KUKA KRL program: edge_1_right_stm.src, edge_1_right_stm.dat

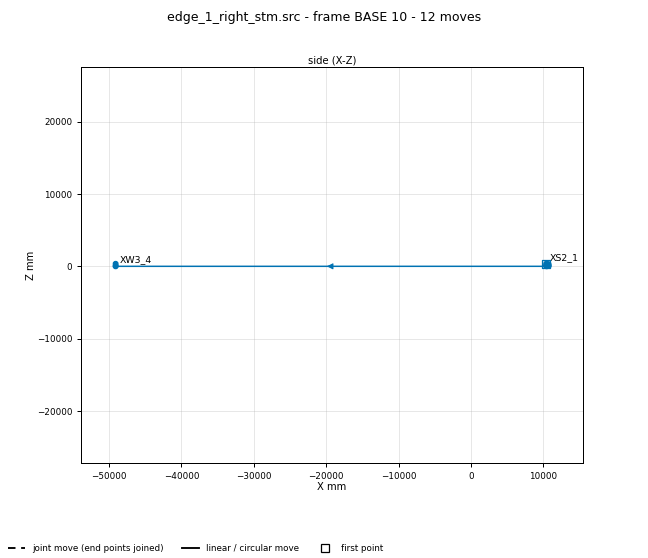
[picture p0: tool path of edge_1_right_stm.src in frame BASE 10, 12 of 12 moves have a stored position in this frame; points joined in program order, loops and branches not executed]
--- edge_1_right_stm.src ---
&ACCESS RVP
&REL 45
&PARAM EDITMASK = *
&PARAM DISKPATH = KRC:\R1\Program
DEF edge_1_right_stm( )
;FOLD INI;%{PE}
  ;FOLD BASISTECH INI
    GLOBAL INTERRUPT DECL 3 WHEN $STOPMESS==TRUE DO IR_STOPM ( )
    INTERRUPT ON 3
    BAS (#INITMOV,0 )
  ;ENDFOLD (BASISTECH INI)
  ;FOLD USER INI
    ;Make your modifications here

  ;ENDFOLD (USER INI)
;ENDFOLD (INI)
TS_CorrOff()
;FOLD PTP S2_1 Vel= 100 % PDATW1_1 Tool[1] Base[10] ;%{PE}%R 8.3.34,%MKUKATPBASIS,%CMOVE,%VPTP,%P 1:PTP, 2:S2_1, 3:C_DIS, 5:100, 7:PDATS2_1
$BWDSTART = FALSE
PDAT_ACT=PPDATS2_1
FDAT_ACT=FS2_1
BAS(#PTP_PARAMS,100)
SET_CD_PARAMS (0)
PTP XS2_1 C_DIS
;ENDFOLD

;FOLD LIN S2_2 Vel= 0.06 m/s CPDATS2_2 TouchSense SEARCH VIA S2_3 CDS2_2 SPS2_2 Tool[1] Base[10] ;%{PE}
;FOLD Parameters ;%{h}
;Params IlfProvider=kukaroboter.touchsense.searchlin; Kuka.PointName=S2_2; Kuka.BlendingEnabled=False; Kuka.MoveDataName=CPDATS2_2; Kuka.VelocityPath=0.06; Kuka.MovementParameterFieldEnabled=True; MoveType=LIN
;FOLD Parameters TouchSense ;%{h}
;Params TouchSense.SearchViaPoint=S2_3;TouchSense.ReferenceMove=CDS2_2;TouchSense.SeachParam=SPS2_2
;ENDFOLD
;ENDFOLD
$BWDSTART = FALSE
LDAT_ACT=LCPDATS2_2
FDAT_ACT=FS2_2
BAS(#CP_PARAMS,0.06)
SET_CD_PARAMS (0)
LIN XS2_2 C_DIS C_DIS
TS_InitMovement($POS_ACT, XS2_3, ZSPS2_2)
TS_ManMoveToVia(XS2_3)
TS_Search(XS2_3, ZSPS2_2, VCDS2_2)
TS_SetCorrData(ZSPS2_2, VCDS2_2)
;ENDFOLD

;FOLD TouchSense Corr 1 CDS2_2;%{E}
;FOLD Parameters Corr 1D ;%{h}
;Params IlfProvider=KukaRoboter.TouchSense.Correction1D;Correction1D=CDS2_2
;ENDFOLD
TS_BC6DCalc(VCDS2_2, TSg_CD0, TSg_CD0, TSg_CD0, TSg_CD0, TSg_CD0)
;ENDFOLD

;FOLD LIN S2_4 Vel= 0.06 m/s CPDATS2_4 TouchSense SEARCH VIA S2_5 CDS2_4 SPS2_4 Tool[1] Base[10] ;%{PE}
;FOLD Parameters ;%{h}
;Params IlfProvider=kukaroboter.touchsense.searchlin; Kuka.PointName=S2_4; Kuka.BlendingEnabled=False; Kuka.MoveDataName=CPDATS2_4; Kuka.VelocityPath=0.06; Kuka.MovementParameterFieldEnabled=True; MoveType=LIN
;FOLD Parameters TouchSense ;%{h}
;Params TouchSense.SearchViaPoint=S2_5;TouchSense.ReferenceMove=CDS2_4;TouchSense.SeachParam=SPS2_4
;ENDFOLD
;ENDFOLD
$BWDSTART = FALSE
LDAT_ACT=LCPDATS2_4
FDAT_ACT=FS2_4
BAS(#CP_PARAMS,0.06)
SET_CD_PARAMS (0)
LIN XS2_4 C_DIS C_DIS
TS_InitMovement($POS_ACT, XS2_5, ZSPS2_4)
TS_ManMoveToVia(XS2_5)
TS_Search(XS2_5, ZSPS2_4, VCDS2_4)
TS_SetCorrData(ZSPS2_4, VCDS2_4)
;ENDFOLD

;FOLD TouchSense Corr 2 CDS2_2 CDS2_4;%{E}
;FOLD Parameters Corr 2D ;%{h}
;Params IlfProvider=KukaRoboter.TouchSense.Correction2D;Correction1D=CDS2_2;Correction2D=CDS2_4
;ENDFOLD
TS_BC6DCalc(VCDS2_2, TSg_CD0, TSg_CD0, VCDS2_4, TSg_CD0, TSg_CD0)
;ENDFOLD

;FOLD LIN S2_6 Vel= 0.06 m/s CPDATS1_2 Tool[1] Base[10] ;%{PE}%R 8.3.34,%MKUKATPBASIS,%CMOVE,%VLIN,%P 1:LIN, 2:S2_6, 3:, 5:0.06, 7:CPDATS2_6
$BWDSTART = FALSE
LDAT_ACT=LCPDATS2_6
FDAT_ACT=FS2_6
BAS(#CP_PARAMS,0.06)
SET_CD_PARAMS (0)
LIN XS2_6 C_DIS C_DIS
;ENDFOLD

;FOLD LIN S2_7 Vel= 0.02 m/s CPDATS2_7 TouchSense SEARCH VIA S2_8 CDS2_7 SPS2_7 Tool[1] Base[10] ;%{PE}
;FOLD Parameters ;%{h}
;Params IlfProvider=kukaroboter.touchsense.searchlin; Kuka.PointName=S2_7; Kuka.BlendingEnabled=False; Kuka.MoveDataName=CPDATS2_7; Kuka.VelocityPath=0.02; Kuka.MovementParameterFieldEnabled=True; MoveType=LIN
;FOLD Parameters TouchSense ;%{h}
;Params TouchSense.SearchViaPoint=S2_8;TouchSense.ReferenceMove=CDS2_7;TouchSense.SeachParam=SPS2_7
;ENDFOLD
;ENDFOLD
$BWDSTART = FALSE
LDAT_ACT=LCPDATS2_7
FDAT_ACT=FS2_7
BAS(#CP_PARAMS,0.02)
SET_CD_PARAMS (0)
LIN XS2_7 C_DIS C_DIS
TS_InitMovement($POS_ACT, XS2_8, ZSPS2_7)
TS_ManMoveToVia(XS2_8)
TS_Search(XS2_8, ZSPS2_7, VCDS2_7)
TS_SetCorrData(ZSPS2_7, VCDS2_7)
;ENDFOLD

;FOLD TouchSense Corr 3 CDS2_2 CDS2_4 CDS2_7;%{E}
;FOLD Parameters Corr 3D ;%{h}
;Params IlfProvider=KukaRoboter.TouchSense.Correction3D;Correction1D=CDS2_2;Correction2D=CDS2_4;Correction3D=CDS2_7
;ENDFOLD
TS_BC6DCalc(VCDS2_2, TSg_CD0, TSg_CD0, VCDS2_4, TSg_CD0, VCDS2_7)
;ENDFOLD

;FOLD LIN S2_9 Vel= 0.1 m/s CPDATS1_2 Tool[1] Base[10] ;%{PE}%R 8.3.34,%MKUKATPBASIS,%CMOVE,%VLIN,%P 1:LIN, 2:S2_9, 3:, 5:0.1, 7:CPDATS2_9
$BWDSTART = FALSE
LDAT_ACT=LCPDATS2_9
FDAT_ACT=FS2_9
BAS(#CP_PARAMS,0.1)
SET_CD_PARAMS (0)
LIN XS2_9 C_DIS C_DIS
;ENDFOLD

;FOLD PTP W3_1 Vel= 100 % PDATW1_1 Tool[1] Base[10] ;%{PE}%R 8.3.34,%MKUKATPBASIS,%CMOVE,%VPTP,%P 1:PTP, 2:W3_1, 3:C_DIS, 5:100, 7:PDATW3_1
$BWDSTART = FALSE
PDAT_ACT=PPDATW3_1
FDAT_ACT=FW3_1
BAS(#PTP_PARAMS,100)
SET_CD_PARAMS (0)
PTP XW3_1 C_DIS
;ENDFOLD

;FOLD LIN W3_2 Vel= 0.2 m/s CPDATS1_2 Tool[1] Base[10] ;%{PE}%R 8.3.34,%MKUKATPBASIS,%CMOVE,%VLIN,%P 1:LIN, 2:W3_2, 3:, 5:0.2, 7:CPDATW3_2
$BWDSTART = FALSE
LDAT_ACT=LCPDATW3_2
FDAT_ACT=FW3_2
BAS(#CP_PARAMS,0.2)
SET_CD_PARAMS (0)
LIN XW3_2 C_DIS C_DIS
;ENDFOLD

custom_sync('hFAFA0000', 'hffff0000', 250)

;FOLD ARCON WDATW3_3 LIN W3_3 Vel= 0.1 m/s CPDATW8_4 Tool[1] Base[10];%{PE}
;FOLD Parameters ;%{h}
;Params IlfProvider=kukaroboter.arctech.arconlin; Kuka.PointName=W3_3; Kuka.BlendingEnabled=False; Kuka.MoveDataName=CPDATW3_3; Kuka.VelocityPath=0.1; Kuka.CurrentCDSetIndex=0; Kuka.MovementParameterFieldEnabled=True; ArcTech.WdatVarName=WDATW3_3
;ENDFOLD
$BWDSTART = FALSE
LDAT_ACT = LCPDATW3_3
FDAT_ACT = FW3_3
BAS(#CP_PARAMS,0.1)
SET_CD_PARAMS (0)
TRIGGER WHEN DISTANCE = 1 DELAY = ArcGetDelay(#PreDefinition, WDATW3_3) DO ArcMainNG(#PreDefinition, WDATW3_3, WW3_3) PRIO = -1
TRIGGER WHEN PATH = ArcGetPath(#OnTheFlyArcOn, WDATW3_3) DELAY = ArcGetDelay(#GasPreflow, WDATW3_3) DO ArcMainNG(#GasPreflow, WDATW3_3, WW3_3) PRIO = -1
TRIGGER WHEN PATH = ArcGetPath(#OnTheFlyArcOn, WDATW3_3) DELAY = 0 DO ArcMainNG(#ArcOnMoveStd, WDATW3_3, WW3_3) PRIO = -1
ArcMainNG(#ArcOnBeforeMoveStd, WDATW3_3, WW3_3)
LIN XW3_3
ArcMainNG(#ArcOnAfterMoveStd, WDATW3_3, WW3_3)
;ENDFOLD

;FOLD ARCOFF WDATW3_4 LIN W3_4 CPDATW3_4 Tool[1] Base[10];%{PE}
;FOLD Parameters ;%{h}
;Params IlfProvider=kukaroboter.arctech.arcofflin; Kuka.IsGlobalPoint=False; Kuka.PointName=W3_4; Kuka.BlendingEnabled=False; Kuka.MoveDataName=CPDATW3_4; Kuka.VelocityPath=0.0063; Kuka.CurrentCDSetIndex=0; Kuka.MovementParameterFieldEnabled=True; ArcTech.WdatVarName=WDATW3_4
;ENDFOLD
$BWDSTART = FALSE
LDAT_ACT = LCPDATW3_4
FDAT_ACT = FW3_4
BAS(#CP_PARAMS, gArcBasVelDefinition)
SET_CD_PARAMS (0)
TRIGGER WHEN PATH = ArcGetPath(#ArcOffBefore, WDATW3_4) DELAY = 0 DO ArcMainNG(#ArcOffBeforeOffStd, WDATW3_4) PRIO = -1
TRIGGER WHEN PATH = ArcGetPath(#OnTheFlyArcOff, WDATW3_4) DELAY = 0 DO ArcMainNG(#ArcOffMoveStd, WDATW3_4) PRIO = -1
ArcMainNG(#ArcOffBeforeMoveStd, WDATW3_4)
LIN XW3_4
ArcMainNG(#ArcOffAfterMoveStd, WDATW3_4)
;ENDFOLD

;FOLD LIN W3_5 Vel= 0.2 m/s CPDATS1_2 Tool[1] Base[10] ;%{PE}%R 8.3.34,%MKUKATPBASIS,%CMOVE,%VLIN,%P 1:LIN, 2:W3_5, 3:, 5:0.2, 7:CPDATW3_5
$BWDSTART = FALSE
LDAT_ACT=LCPDATW3_5
FDAT_ACT=FW3_5
BAS(#CP_PARAMS,0.2)
SET_CD_PARAMS (0)
LIN XW3_5 C_DIS C_DIS
;ENDFOLD

;FOLD LIN W3_6 Vel= 0.4 m/s CPDATS1_2 Tool[1] Base[10] ;%{PE}%R 8.3.34,%MKUKATPBASIS,%CMOVE,%VLIN,%P 1:LIN, 2:W3_6, 3:, 5:0.4, 7:CPDATW3_6
$BWDSTART = FALSE
LDAT_ACT=LCPDATW3_6
FDAT_ACT=FW3_6
BAS(#CP_PARAMS,0.4)
SET_CD_PARAMS (0)
LIN XW3_6 C_DIS C_DIS
;ENDFOLD

TS_CorrOff()
ochistka_mod()
END

--- edge_1_right_stm.dat ---
&ACCESS RVP
&REL 45
&PARAM EDITMASK = *
&PARAM DISKPATH = KRC:\R1\Program
DEFDAT  edge_1_right_stm
;FOLD EXTERNAL DECLARATIONS;%{PE}%MKUKATPBASIS,%CEXT,%VCOMMON,%P
;FOLD BASISTECH EXT;%{PE}%MKUKATPBASIS,%CEXT,%VEXT,%P
EXT  BAS (BAS_COMMAND  :IN,REAL  :IN )
DECL INT SUCCESS
;ENDFOLD (BASISTECH EXT)
;FOLD USER EXT;%{E}%MKUKATPUSER,%CEXT,%VEXT,%P
;Make your modifications here

;ENDFOLD (USER EXT)
;ENDFOLD (EXTERNAL DECLARATIONS)

DECL PDAT PPDATS2_1={VEL 100,ACC 100.0,APO_DIST 10.0,GEAR_JERK 50.0000,EXAX_IGN 0}
DECL FDAT FS2_1={TOOL_NO 1,BASE_NO 10,IPO_FRAME #BASE,POINT2[] " "}
DECL E6POS XS2_1={X 10410.0,Y 968.0,Z 366.0,A -120,B 50,C -180,S 20,T 53,E1 9363.166987703404,E2 0,E3 465.0,E4 0,E5 0,E6 0}

DECL E6POS XS2_2={X 10410.0,Y 968.0,Z 76.0,A -120,B 50,C -180,S 20,T 53,E1 9363.166987703404,E2 0,E3 465.0,E4 0,E5 0,E6 0}
DECL FDAT FS2_2={TOOL_NO 1,BASE_NO 10,IPO_FRAME #BASE,POINT2[] " ",TQ_STATE FALSE}
DECL LDAT LCPDATS2_2={VEL 0.06,ACC 100.0,APO_DIST 10.0,APO_FAC 50.0,ORI_TYP #VAR,CIRC_TYP #BASE,JERK_FAC 50.0}
DECL E6POS XS2_3={X 10410.0,Y 968.0,Z 16.0,A -120,B 50,C -180,S 20,T 53,E1 9363.166987703404,E2 0,E3 465.0,E4 0,E5 0,E6 0}
DECL FDAT FS2_3={TOOL_NO 1,BASE_NO 10,IPO_FRAME #BASE,POINT2[] " ",TQ_STATE FALSE}
DECL TSg_PCollCD_T VCDS2_2={CD_IPO_MODE #BASE,Mastered TRUE,SDir_W {X 0.0,Y 0.0,Z 0.0,A 0.0,B 0.0,C 0.0},Ref_W {X 10410.0,Y 968.0,Z 16.0,A -120,B 50,C -180},Meas_W {X 0.0,Y 0.0,Z 0.0,A 0.0,B 0.0,C 0.0},Diff_W {X 0.0,Y 0.0,Z 0.0,A 0.0,B 0.0,C 0.0},VecLenDiff_W 0.0,MEnum #CDEmpty,MC 1}
DECL TSg_SearchProperty_T ZSPS2_2={MoveType #MoveWithLin,TouchType #Single,DynamicStep #Slow,SensorNum 1,SearchDepth_Tol 150.0,bBackToStartPos TRUE}

DECL E6POS XS2_4={X 10410.0,Y 968.0,Z 76.0,A -120,B 50,C 169,S 20,T 53,E1 9416.675227415548,E2 0,E3 465.0,E4 0,E5 0,E6 0}
DECL FDAT FS2_4={TOOL_NO 1,BASE_NO 10,IPO_FRAME #BASE,POINT2[] " ",TQ_STATE FALSE}
DECL LDAT LCPDATS2_4={VEL 0.06,ACC 100.0,APO_DIST 10.0,APO_FAC 50.0,ORI_TYP #VAR,CIRC_TYP #BASE,JERK_FAC 50.0}
DECL E6POS XS2_5={X 10410.0,Y 908.0,Z 76.0,A -120,B 50,C 169,S 20,T 53,E1 9416.675227415548,E2 0,E3 465.0,E4 0,E5 0,E6 0}
DECL FDAT FS2_5={TOOL_NO 1,BASE_NO 10,IPO_FRAME #BASE,POINT2[] " ",TQ_STATE FALSE}
DECL TSg_PCollCD_T VCDS2_4={CD_IPO_MODE #BASE,Mastered TRUE,SDir_W {X 0.0,Y 0.0,Z 0.0,A 0.0,B 0.0,C 0.0},Ref_W {X 10410.0,Y 908.0,Z 76.0,A -120,B 50,C 169},Meas_W {X 0.0,Y 0.0,Z 0.0,A 0.0,B 0.0,C 0.0},Diff_W {X 0.0,Y 0.0,Z 0.0,A 0.0,B 0.0,C 0.0},VecLenDiff_W 0.0,MEnum #CDEmpty,MC 1}
DECL TSg_SearchProperty_T ZSPS2_4={MoveType #MoveWithLin,TouchType #Single,DynamicStep #Slow,SensorNum 1,SearchDepth_Tol 150.0,bBackToStartPos TRUE}

DECL LDAT LCPDATS2_6={VEL 0.06,ACC 100.0,APO_DIST 10.0,APO_FAC 50.0,ORI_TYP #VAR,CIRC_TYP #BASE,JERK_FAC 50.0,GEAR_JERK 50.0000,EXAX_IGN 0}
DECL FDAT FS2_6={TOOL_NO 1,BASE_NO 10,IPO_FRAME #BASE,POINT2[] " "}
DECL E6POS XS2_6={X 10730.0,Y 968.0,Z 76.0,A -120,B 40,C -169,S 20,T 53,E1 9689.593440362198,E2 0,E3 465.0,E4 0,E5 0,E6 0}

DECL E6POS XS2_7={X 10730.0,Y 898.0,Z 76.0,A -120,B 40,C -169,S 20,T 53,E1 9689.593440362198,E2 0,E3 465.0,E4 0,E5 0,E6 0}
DECL FDAT FS2_7={TOOL_NO 1,BASE_NO 10,IPO_FRAME #BASE,POINT2[] " ",TQ_STATE FALSE}
DECL LDAT LCPDATS2_7={VEL 0.02,ACC 100.0,APO_DIST 10.0,APO_FAC 50.0,ORI_TYP #VAR,CIRC_TYP #BASE,JERK_FAC 50.0}
DECL E6POS XS2_8={X 10670.0,Y 898.0,Z 76.0,A -120,B 40,C -169,S 20,T 53,E1 9689.593440362198,E2 0,E3 465.0,E4 0,E5 0,E6 0}
DECL FDAT FS2_8={TOOL_NO 1,BASE_NO 10,IPO_FRAME #BASE,POINT2[] " ",TQ_STATE FALSE}
DECL TSg_PCollCD_T VCDS2_7={CD_IPO_MODE #BASE,Mastered TRUE,SDir_W {X 0.0,Y 0.0,Z 0.0,A 0.0,B 0.0,C 0.0},Ref_W {X 10670.0,Y 898.0,Z 76.0,A -120,B 40,C -169},Meas_W {X 0.0,Y 0.0,Z 0.0,A 0.0,B 0.0,C 0.0},Diff_W {X 0.0,Y 0.0,Z 0.0,A 0.0,B 0.0,C 0.0},VecLenDiff_W 0.0,MEnum #CDEmpty,MC 1}
DECL TSg_SearchProperty_T ZSPS2_7={MoveType #MoveWithLin,TouchType #Single,DynamicStep #Slow,SensorNum 1,SearchDepth_Tol 150.0,bBackToStartPos TRUE}

DECL LDAT LCPDATS2_9={VEL 0.1,ACC 100.0,APO_DIST 10.0,APO_FAC 50.0,ORI_TYP #VAR,CIRC_TYP #BASE,JERK_FAC 50.0,GEAR_JERK 50.0000,EXAX_IGN 0}
DECL FDAT FS2_9={TOOL_NO 1,BASE_NO 10,IPO_FRAME #BASE,POINT2[] " "}
DECL E6POS XS2_9={X 10730.0,Y 968.0,Z 316.0,A -150,B 50,C -169,S 20,T 53,E1 9713.992948913843,E2 0,E3 465.0,E4 0,E5 0,E6 0}

DECL PDAT PPDATW3_1={VEL 100,ACC 100.0,APO_DIST 10.0,GEAR_JERK 50.0000,EXAX_IGN 0}
DECL FDAT FW3_1={TOOL_NO 1,BASE_NO 10,IPO_FRAME #BASE,POINT2[] " "}
DECL E6POS XW3_1={X 10467.0,Y 968.0,Z 366.0,A -118.5,B 41.3,C 160.3,S 20,T 53,E1 9761.697010935082,E2 0,E3 465.0,E4 0,E5 0,E6 0}

DECL LDAT LCPDATW3_2={VEL 0.2,ACC 100.0,APO_DIST 10.0,APO_FAC 50.0,ORI_TYP #VAR,CIRC_TYP #BASE,JERK_FAC 50.0,GEAR_JERK 50.0000,EXAX_IGN 0}
DECL FDAT FW3_2={TOOL_NO 1,BASE_NO 10,IPO_FRAME #BASE,POINT2[] " "}
DECL E6POS XW3_2={X 10467.0,Y 968.0,Z 76.0,A -118.5,B 41.3,C 160.3,S 20,T 53,E1 9761.697010935082,E2 0,E3 465.0,E4 0,E5 0,E6 0}

DECL stArcDat_T WDATW3_3={Strike {JobModeId[] "Job Mode",ParamSetId[] "Set1",StartTime 0.0,PreFlowTime 0.0,Channel1 1,Channel2 0.0,Channel3 0.0,Channel4 0.0,Channel5 0.0,Channel6 0.0,Channel7 0.0,Channel8 0.0,PurgeTime 0.0},Weld {JobModeId[] "Job Mode",ParamSetId[] "Set2",Velocity 0.0063,Channel1 1,Channel2 0,Channel3 0.0,Channel4 0.0,Channel5 0.0,Channel6 0.0,Channel7 0.0,Channel8 0.0},Weave {Pattern #Triangle,Length 3.5,Amplitude 2,Angle 0.0,LeftSideDelay 0.0,RightSideDelay 0.0},Advanced {IgnitionErrorStrategy 1,WeldErrorStrategy 1,SlopeOption #None,SlopeTime 0.0,SlopeDistance 0.0,OnTheFlyActiveOn FALSE,OnTheFlyActiveOff FALSE,OnTheFlyDistanceOn 0.0,OnTheFlyDistanceOff 0.0},Track {IsArcSenseEnabled TRUE,ControlEnabled TRUE,KeepOffset TRUE,TeachNew FALSE,FindSeamMiddle TRUE,TrackingDelay 0.2,ControlSensibility 25.0,MaxDeviation 100,ControlSensibilityHeight 25.0,Bias 0.0,WeaveOffset 0.0,HeightCorrValue 0.0}}
DECL stArcDat_T WW3_3={Strike {SeamName[] " ",SeamNumber -1},Advanced {BitCodedRobotMark 0}}
DECL E6POS XW3_3={X 10467.0,Y 908.0,Z 16.0,A -118.5,B 41.3,C 160.3,S 20,T 53,E1 9761.697010935082,E2 0,E3 405.0,E4 0,E5 0,E6 0}
DECL FDAT FW3_3={TOOL_NO 1,BASE_NO 10,IPO_FRAME #BASE,POINT2[] " "}
DECL LDAT LCPDATW3_3={VEL 0.1,ACC 100.0,APO_DIST 0.0,APO_FAC 50.0,AXIS_VEL 100.0,AXIS_ACC 100.0,ORI_TYP #VAR,CIRC_TYP #BASE,JERK_FAC 50.0,GEAR_JERK 50.0,EXAX_IGN 0}

DECL stArcDat_T WDATW3_4={Crater {JobModeId[] "Job Mode",ParamSetId[] "Set3",CraterTime 0.0,PostflowTime 0.0,Channel1 1,Channel2 0.0,Channel3 0.0,Channel4 0.0,Channel5 0.0,Channel6 0.0,Channel7 0.0,Channel8 0.0,BurnBackTime 0.0},Advanced {IgnitionErrorStrategy 1,WeldErrorStrategy 1,SlopeOption #None,SlopeTime 0.0,SlopeDistance 0.0,OnTheFlyActiveOn FALSE,OnTheFlyActiveOff FALSE,OnTheFlyDistanceOn 0.0,OnTheFlyDistanceOff 0.0}}
DECL E6POS XW3_4={X -49080.0,Y 908.0,Z 15.0,A -118.5,B 41.3,C 160.3,S 20,T 53,E1 -10000,E2 0,E3 405.0,E4 0,E5 0,E6 0}
DECL FDAT FW3_4={TOOL_NO 1,BASE_NO 10,IPO_FRAME #BASE,POINT2[] " "}
DECL LDAT LCPDATW3_4={VEL 0.01,ACC 100.0,APO_DIST 0.0,APO_FAC 50.0,AXIS_VEL 100.0,AXIS_ACC 100.0,ORI_TYP #VAR,CIRC_TYP #BASE,JERK_FAC 50.0,GEAR_JERK 50.0,EXAX_IGN 0}

DECL LDAT LCPDATW3_5={VEL 0.2,ACC 100.0,APO_DIST 10.0,APO_FAC 50.0,ORI_TYP #VAR,CIRC_TYP #BASE,JERK_FAC 50.0,GEAR_JERK 50.0000,EXAX_IGN 0}
DECL FDAT FW3_5={TOOL_NO 1,BASE_NO 10,IPO_FRAME #BASE,POINT2[] " "}
DECL E6POS XW3_5={X -49080.0,Y 968.0,Z 75.0,A -118.5,B 41.3,C 160.3,S 20,T 53,E1 -10000,E2 0,E3 465.0,E4 0,E5 0,E6 0}

DECL LDAT LCPDATW3_6={VEL 0.4,ACC 100.0,APO_DIST 10.0,APO_FAC 50.0,ORI_TYP #VAR,CIRC_TYP #BASE,JERK_FAC 50.0,GEAR_JERK 50.0000,EXAX_IGN 0}
DECL FDAT FW3_6={TOOL_NO 1,BASE_NO 10,IPO_FRAME #BASE,POINT2[] " "}
DECL E6POS XW3_6={X -49080.0,Y 968.0,Z 365.0,A -118.5,B 41.3,C 160.3,S 20,T 53,E1 -10000,E2 0,E3 465.0,E4 0,E5 0,E6 0}
ENDDAT
